FUNCTION_BLOCK FB_Valve_2_10V IMPLEMENTS I_Valve
VAR_INPUT
END_VAR
VAR_OUTPUT
END_VAR
VAR
	//Properties
	bError : BOOL := FALSE;
	fOpeningActual : REAL;
	fOpeningSetpoint : REAL := 0;
	//Raw values
	nOpeningSet AT %Q* : INT;
	nOpeningAct AT %I* : INT;
END_VAR

PROPERTY Error : BOOL
GET
Error := THIS^.bError;
END_GET
SET
THIS^.bError := Error;
END_SET
END_PROPERTY

PROPERTY OpeningActual : REAL
GET
OpeningActual := THIS^.fOpeningActual;
END_GET
SET
THIS^.fOpeningActual := OpeningActual;
END_SET
END_PROPERTY

PROPERTY OpeningSetpoint : REAL
GET
OpeningSetpoint := THIS^.fOpeningSetpoint;
END_GET
SET
THIS^.fOpeningSetpoint := OpeningSetpoint;
END_SET
END_PROPERTY

METHOD Run
//Read feedback for opening position
fOpeningActual := FC_Voltage2_10Raw_TO_Percentage(nOpeningAct);

//Write setpoint for opening position
nOpeningSet := FC_Percentage_TO_Voltage2_10Raw(fOpeningSetpoint);
END_METHOD

END_FUNCTION_BLOCK

(* stored: Version 1.1.0.1, ProductVersion 3.1.4024.0
   POU FB_Valve_2_10V: Id {641d499c-e925-4856-a53e-eb0195b38f06}, SpecialFunc None
   Property Error: Id {af0ab811-355e-449d-9952-1cf62d68eaee}
   Get Get: Id {404e7f5b-a288-4a60-8ce5-de5731bdc574}
   Set Set: Id {edb892bd-b7f0-473e-bfca-5bbb37b7542c}
   Property OpeningActual: Id {55a91989-1b4c-4ecf-8e56-7eee0efb99ad}
   Get Get: Id {0d9ac439-ce16-40ad-b688-090cba006d4e}
   Set Set: Id {c2b3162a-3400-40d8-b74e-7ba09b47fe57}
   Property OpeningSetpoint: Id {78602e66-cd35-4c54-829b-fcf79cefa1d0}
   Get Get: Id {4b19c777-324b-40b4-be02-c49b458a48f8}
   Set Set: Id {910197a3-50e8-4831-b4a7-cff369bebf57}
   Method Run: Id {4bfa6015-a7e4-47e7-8694-71b44d8c0622} *)
